(* CODESYS project maquinaDeLavar.project

Project tree, tasks and I/O mapping:
  Device : CODESYS Control Win V3, 3S - Smart Software Solutions GmbH, order no. 305021, version 3.5.11.30
    application Application
      libraries: Standard, * (System)
      task MainTask (cyclic, interval t#20ms, priority 1) calls PLC_PRG
      program PLC_PRG [SFC]: P0_active, P1_active, P4_active, P5_active, P6_active, P7_active, T8_active, T9_active, T10_active, T11_active, T12_active, T8_entry, T12_entry, P3_active, P3_active_0
*)

// Device/Application/PLC_PRG
PROGRAM PLC_PRG
VAR
	// LIGAR
	B1: BOOL;
	B2: BOOL;
	
	NIVEL: INT;
	BN3: BOOL; //SELECIONA O PROGRAMA DE LV
	BN5: BOOL;
	BN10: BOOL;
	
	ENXAGUES: INT;
	EN1: BOOL; //SELECIONA O NUERO DE ENXAGUES
	EN2: BOOL;
	EN3: BOOL;
	
	PF:BOOL; //SENSOR DA PORTA
	V1: BOOL; //VALVULA AGUA
	V2: BOOL; //VALVULA SABAO
	V3: BOOL; //VALVULA DESCARTE DA AGUA
	
	
	P: REAL; //SENSOR DE NIVEL
	T: REAL; //SENSOR DE TEMPERATURA
	
	KM3: BOOL; //CONTATOR DO MOTOR SENTIDO INVERSO
	KR: BOOL; //CONTATOR DA RESISTNCIA
	KM1: BOOL; //CONTATOR DO MOTOR SENTIDO NORMAL
	KM2: BOOL;
	
	CONT: INT;
END_VAR

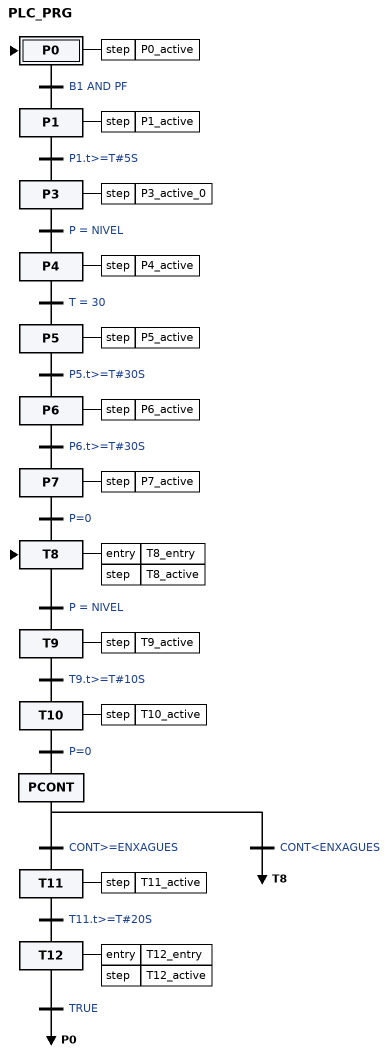
INITIAL_STEP P0:
    P0_active(N);  // step action
END_STEP
TRANSITION FROM P0 TO P1
    := B1 AND PF;
END_TRANSITION
STEP P1:
    P1_active(N);  // step action
END_STEP
TRANSITION FROM P1 TO P3
    := P1.t>=T#5S;
END_TRANSITION
STEP P3:
    P3_active_0(N);  // step action
END_STEP
TRANSITION FROM P3 TO P4
    := P = NIVEL;
END_TRANSITION
STEP P4:
    P4_active(N);  // step action
END_STEP
TRANSITION FROM P4 TO P5
    := T = 30;
END_TRANSITION
STEP P5:
    P5_active(N);  // step action
END_STEP
TRANSITION FROM P5 TO P6
    := P5.t>=T#30S;
END_TRANSITION
STEP P6:
    P6_active(N);  // step action
END_STEP
TRANSITION FROM P6 TO P7
    := P6.t>=T#30S;
END_TRANSITION
STEP P7:
    P7_active(N);  // step action
END_STEP
TRANSITION FROM P7 TO T8
    := P=0;
END_TRANSITION
STEP T8:
    T8_entry(P1);  // entry action
    T8_active(N);  // step action
END_STEP
TRANSITION FROM T8 TO T9
    := P = NIVEL;
END_TRANSITION
STEP T9:
    T9_active(N);  // step action
END_STEP
TRANSITION FROM T9 TO T10
    := T9.t>=T#10S;
END_TRANSITION
STEP T10:
    T10_active(N);  // step action
END_STEP
TRANSITION FROM T10 TO PCONT
    := P=0;
END_TRANSITION
STEP PCONT:
END_STEP
TRANSITION FROM PCONT TO T11
    := CONT>=ENXAGUES;
END_TRANSITION
TRANSITION FROM PCONT TO T8
    := CONT<ENXAGUES;
END_TRANSITION
STEP T11:
    T11_active(N);  // step action
END_STEP
TRANSITION FROM T11 TO T12
    := T11.t>=T#20S;
END_TRANSITION
STEP T12:
    T12_entry(P1);  // entry action
    T12_active(N);  // step action
END_STEP
TRANSITION FROM T12 TO P0
    := TRUE;
END_TRANSITION

ACTION P0_active:
IF BN3 THEN 
	NIVEL:= 3;
END_IF

IF BN5 THEN 
	NIVEL:= 5;
END_IF

IF BN10 THEN 
	NIVEL:= 10;
END_IF


IF EN1 THEN 
	ENXAGUES:= 1;
END_IF

IF EN2 THEN 
	ENXAGUES:= 2;
END_IF

IF EN3 THEN 
	ENXAGUES:= 3;
END_IF
END_ACTION

ACTION P1_active:
V1:=TRUE;
V2:=TRUE;
END_ACTION

ACTION P4_active:
V2:= FALSE;
V1:= FALSE;
KM3:= TRUE;
KR:= TRUE;
END_ACTION

ACTION P5_active:
KM3:= FALSE;
KR:= FALSE;
END_ACTION

ACTION P6_active:
KM1:= TRUE;
END_ACTION

ACTION P7_active:
KM1:=FALSE;
V3:= TRUE;
END_ACTION

ACTION T8_active:
V1:=TRUE;
V3:=FALSE;
END_ACTION

ACTION T9_active:
KM3:= TRUE;
V1:=FALSE;
END_ACTION

ACTION T10_active:
KM3:= FALSE;
V3:=TRUE;
END_ACTION

ACTION T11_active:
V3:=TRUE;
KM2:= TRUE;
END_ACTION

ACTION T12_active:
V3:=FALSE;
KM2:= FALSE;
END_ACTION

ACTION T8_entry:
CONT:=CONT+1;
END_ACTION

ACTION T12_entry:
CONT:= 0;
END_ACTION

ACTION P3_active:
V2:=FALSE;
END_ACTION

ACTION P3_active_0:
V2:=FALSE;
END_ACTION

END_PROGRAM
